FUNCTION_BLOCK FB_PowerAll
VAR_INPUT
	Enable 		: BOOL;
END_VAR
VAR_IN_OUT
	acs: ARRAY[1..6] OF AXIS_REF;
	mcs: ARRAY[1..6] OF AXIS_REF;
END_VAR
VAR_OUTPUT
	Status		: BOOL;
	Error		: BOOL;
END_VAR
VAR
	fbPower 	: ARRAY [1..12] OF MC_Power;
	i			: UINT;
END_VAR

Status := TRUE;
Error := FALSE;

FOR i:=1 TO 6 DO
	
	fbPower[i](
		Axis:= acs[i], 
		Enable:= Enable, 
		Enable_Positive:= Enable, 
		Enable_Negative:= Enable, 
		Override:= , 
		BufferMode:= MC_BufferMode.MC_Buffered, 
		Options:= , 
		Status=> , 
		Busy=> , 
		Error=> , 
		ErrorID=> );
		
	fbPower[i+6](
		Axis:= mcs[i], 
		Enable:= Enable, 
		Enable_Positive:= Enable, 
		Enable_Negative:= Enable, 
		Override:= , 
		BufferMode:= MC_BufferMode.MC_Buffered, 
		Options:= , 
		Status=> , 
		Busy=> , 
		Error=> , 
		ErrorID=> );
	
	Status := Status AND fbPower[i].Status AND fbPower[i+6].Status; 
	Error := Error OR fbPower[i].Error OR fbPower[i+6].Error;
	
END_FOR

END_FUNCTION_BLOCK

(* stored: Version 1.1.0.1
   POU FB_PowerAll: Id {d3e6d2d4-b215-4a84-8022-bf06b4a82234}, SpecialFunc None *)
